{attribute 'no_explicit_call' := 'do not call this POU directly'} 
FUNCTION_BLOCK VFD
VAR
END_VAR

METHOD executeOperation : BOOL
VAR_INPUT
	SpeedRel 	: LREAL;
	TorqueRel	: LREAL;
END_VAR
END_METHOD

PROPERTY Speed : LREAL
GET
END_GET
END_PROPERTY

PROPERTY SpeedMax : LREAL
GET
END_GET
END_PROPERTY

PROPERTY Torque : LREAL
GET
END_GET
END_PROPERTY

PROPERTY TorqueMax : LREAL
GET
END_GET
END_PROPERTY

PROPERTY TorqueRel : LREAL
GET
END_GET
END_PROPERTY

METHOD update : BOOL
VAR_INPUT
END_VAR
END_METHOD

END_FUNCTION_BLOCK

(* stored: Version 1.1.0.1
   POU VFD: Id {16d0b88d-bfb7-0c59-06c6-71c8d1f37c47}, SpecialFunc None
   Method executeOperation: Id {99cbc759-9fc9-0ce6-0a30-d4d6060afe93}
   Property Speed: Id {85d64c6f-c52c-099d-1fed-ed6c3b464301}
   Get Get: Id {f250d892-8c10-0a4c-2959-c6230b4068cc}
   Property SpeedMax: Id {d3a98068-0031-06b8-2da9-1feeff214ce1}
   Get Get: Id {ed7e69d1-e98e-0d66-3e17-f213c69b0b99}
   Property Torque: Id {1dbc2f31-654a-073b-14bf-b792193a2c99}
   Get Get: Id {f9be3ff2-398b-00c1-184a-b8db285a4dc7}
   Property TorqueMax: Id {ddbe2a83-ce23-0310-351f-52e096aa2538}
   Get Get: Id {5ab459a4-0d87-0512-3f39-f9564b2d3acf}
   Property TorqueRel: Id {2968dfc1-041d-022f-00fe-6a02e2f262d4}
   Get Get: Id {2d7e146c-bd78-0602-2369-6dd386bf1236}
   Method update: Id {cedb65b2-7991-05f7-2a0d-0e66b4975d69} *)
